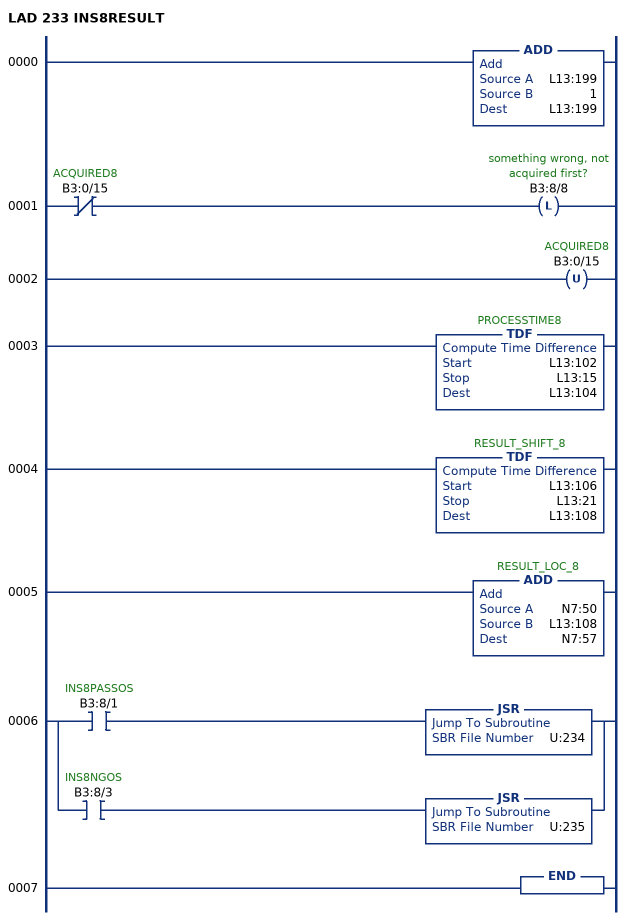
% Rung: 0 %
SOR ADD L13:199 1 L13:199 EOR
% Rung: 1 %
SOR XIO B3:0/15 OTL B3:8/8 EOR
%   B3:0/15  ACQUIRED8 %
%   B3:8/8  "something wrong, not acquired first?" %
% Rung: 2 %
SOR OTU B3:0/15 EOR
%   B3:0/15  ACQUIRED8 %
% Rung: 3 %
SOR TDF L13:102 L13:15 L13:104 EOR
%   L13:102  TIMEOFACQ8 %
%   L13:15  TOP_TIME %
%   L13:104  PROCESSTIME8 %
% Rung: 4 %
SOR TDF L13:106 L13:21 L13:108 EOR
%   L13:106  PROCESS_START_POS_8 %
%   L13:21  TOP_POSITION %
%   L13:108  RESULT_SHIFT_8 %
% Rung: 5 %
SOR ADD N7:50 L13:108 N7:57 EOR
%   N7:50  INS_8_TRIG_LOC %
%   L13:108  RESULT_SHIFT_8 %
%   N7:57  RESULT_LOC_8 %
% Rung: 6 %
SOR BST XIC B3:8/1 JSR U:234 NXB XIC B3:8/3 JSR U:235 BND EOR
%   B3:8/1  INS8PASSOS %
%   B3:8/3  INS8NGOS %
% Rung: 7 %
SOR END EOR

LADDER 234 "INS8PASS"
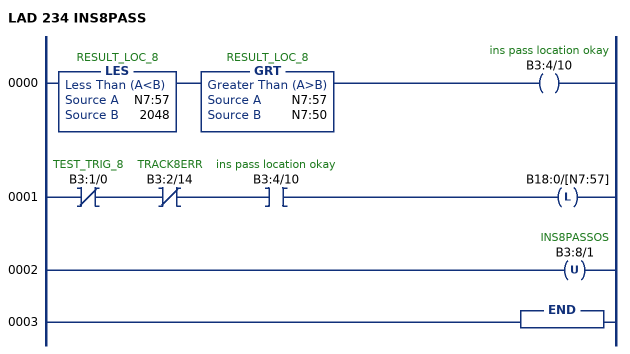
% Rung: 0 %
SOR LES N7:57 2048 GRT N7:57 N7:50 OTE B3:4/10 EOR
%   N7:57  RESULT_LOC_8 %
%   N7:50  INS_8_TRIG_LOC %
%   B3:4/10  "ins pass location okay" %
% Rung: 1 %
SOR XIO B3:1/0 XIO B3:2/14 XIC B3:4/10 OTL B18:0/[N7:57] EOR
%   B3:1/0  TEST_TRIG_8 %
%   B3:2/14  TRACK8ERR %
%   B3:4/10  "ins pass location okay" %
%   B18:0  GOOD2 %
%   N7:57  RESULT_LOC_8 %
% Rung: 2 %
SOR OTU B3:8/1 EOR
%   B3:8/1  INS8PASSOS %
% Rung: 3 %
SOR END EOR

LADDER 235 "INS8FAIL"
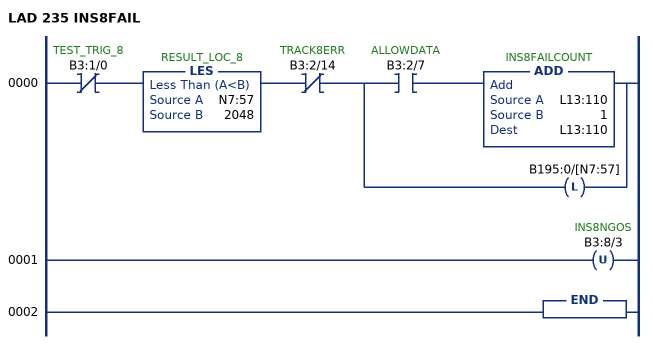
% Rung: 0 %
SOR XIO B3:1/0 LES N7:57 2048 XIO B3:2/14 BST XIC B3:2/7 ADD L13:110 1 L13:110 NXB OTL B195:0/[N7:57] BND EOR
%   B3:1/0  TEST_TRIG_8 %
%   N7:57  RESULT_LOC_8 %
%   B3:2/14  TRACK8ERR %
%   B3:2/7  ALLOWDATA %
%   L13:110  INS8FAILCOUNT %
%   B195:0  TOP_NG %
% Rung: 1 %
SOR OTU B3:8/3 EOR
%   B3:8/3  INS8NGOS %
% Rung: 2 %
SOR END EOR

LADDER 236 "INS8ACQ"
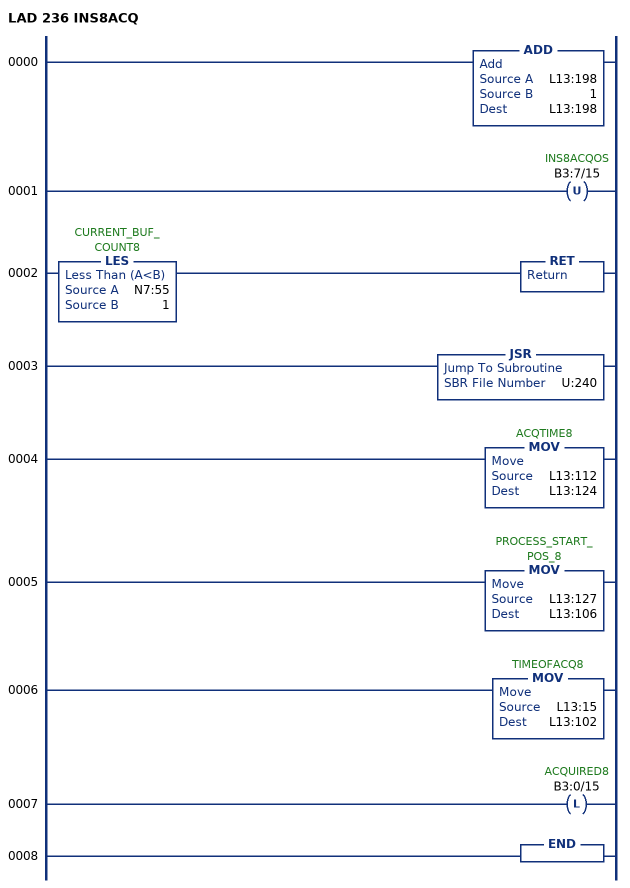
% Rung: 0 %
SOR ADD L13:198 1 L13:198 EOR
% Rung: 1 %
SOR OTU B3:7/15 EOR
%   B3:7/15  INS8ACQOS %
% Rung: 2 %
SOR LES N7:55 1 RET EOR
%   N7:55  CURRENT_BUF_COUNT8 %
% Rung: 3 %
SOR JSR U:240 EOR
% Rung: 4 %
SOR MOV L13:112 L13:124 EOR
%   L13:112  TIME_SPAN8 %
%   L13:124  ACQTIME8 %
% Rung: 5 %
SOR MOV L13:127 L13:106 EOR
%   L13:127  PULLED_POSITION8 %
%   L13:106  PROCESS_START_POS_8 %
% Rung: 6 %
SOR MOV L13:15 L13:102 EOR
%   L13:15  TOP_TIME %
%   L13:102  TIMEOFACQ8 %
% Rung: 7 %
SOR OTL B3:0/15 EOR
%   B3:0/15  ACQUIRED8 %
% Rung: 8 %
SOR END EOR

LADDER 237 "Q8TIMETEST"
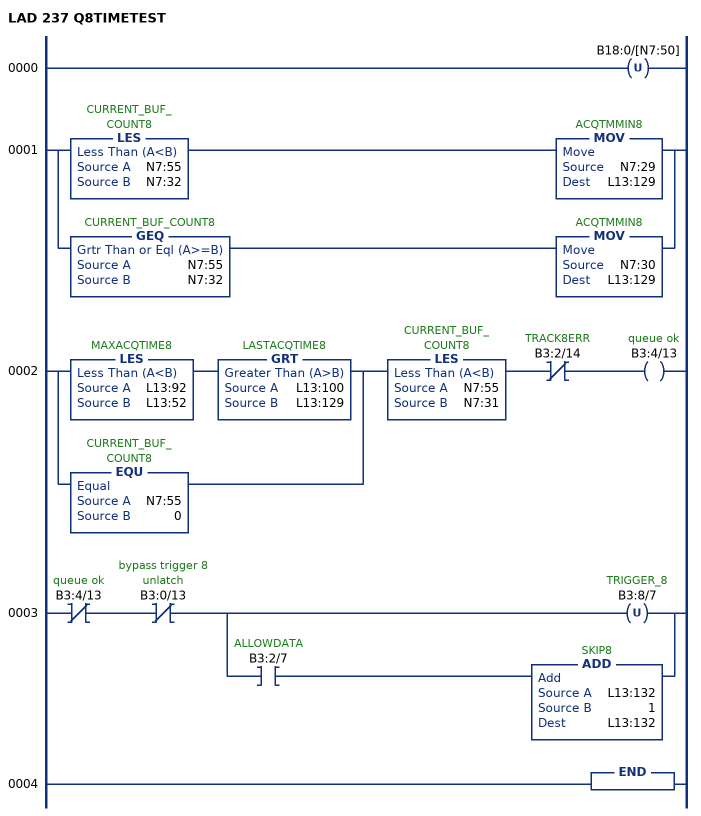
% Rung: 0 %
SOR OTU B18:0/[N7:50] EOR
%   B18:0  GOOD2 %
%   N7:50  INS_8_TRIG_LOC %
% Rung: 1 %
SOR BST LES N7:55 N7:32 MOV N7:29 L13:129 NXB GEQ N7:55 N7:32 MOV N7:30 L13:129 BND EOR
%   N7:55  CURRENT_BUF_COUNT8 %
%   N7:32  BUF_CAM_LIMIT %
%   N7:29  CAM_BUF_ACQ_TM %
%   L13:129  ACQTMMIN8 %
%   N7:30  PC_BUF_ACQ_TM %
% Rung: 2 %
SOR BST LES L13:92 L13:52 GRT L13:100 L13:129 NXB EQU N7:55 0 BND LES N7:55 N7:31 XIO B3:2/14 OTE B3:4/13 EOR
%   L13:92  MAXACQTIME8 %
%   L13:52  ACQTIMELIMIT %
%   L13:100  LASTACQTIME8 %
%   L13:129  ACQTMMIN8 %
%   N7:55  CURRENT_BUF_COUNT8 %
%   N7:31  MAX_BUFF_CT  "maximum buffers" %
%   B3:2/14  TRACK8ERR %
%   B3:4/13  "queue ok" %
% Rung: 3 %
SOR XIO B3:4/13 XIO B3:0/13 BST OTU B3:8/7 NXB XIC B3:2/7 ADD L13:132 1 L13:132 BND EOR
%   B3:4/13  "queue ok" %
%   B3:0/13  "bypass trigger 8 unlatch" %
%   B3:8/7  TRIGGER_8 %
%   B3:2/7  ALLOWDATA %
%   L13:132  SKIP8 %
% Rung: 4 %
SOR END EOR

LADDER 238 "INS8TRIG"
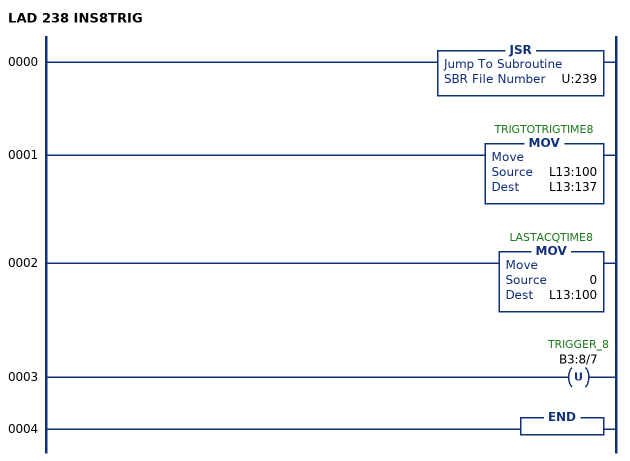
% Rung: 0 %
SOR JSR U:239 EOR
% Rung: 1 %
SOR MOV L13:100 L13:137 EOR
%   L13:100  LASTACQTIME8 %
%   L13:137  TRIGTOTRIGTIME8 %
% Rung: 2 %
SOR MOV 0 L13:100 EOR
%   L13:100  LASTACQTIME8 %
% Rung: 3 %
SOR OTU B3:8/7 EOR
%   B3:8/7  TRIGGER_8 %
% Rung: 4 %
SOR END EOR

LADDER 239 "FIFO8SET"
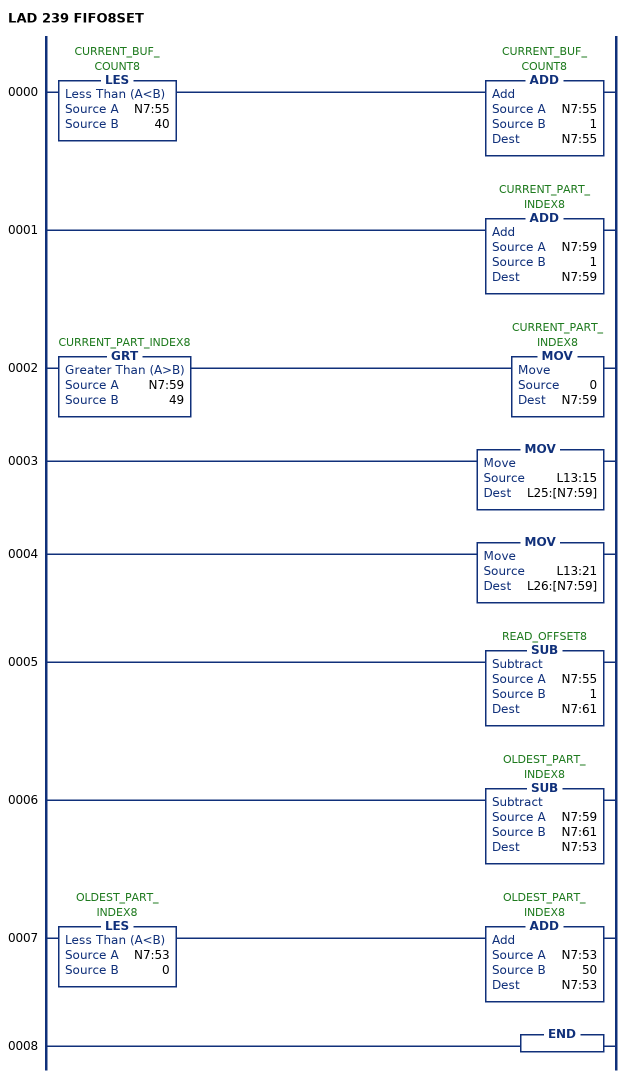
% Rung: 0 %
SOR LES N7:55 40 ADD N7:55 1 N7:55 EOR
%   N7:55  CURRENT_BUF_COUNT8 %
% Rung: 1 %
SOR ADD N7:59 1 N7:59 EOR
%   N7:59  CURRENT_PART_INDEX8 %
% Rung: 2 %
SOR GRT N7:59 49 MOV 0 N7:59 EOR
%   N7:59  CURRENT_PART_INDEX8 %
% Rung: 3 %
SOR MOV L13:15 L25:[N7:59] EOR
%   L13:15  TOP_TIME %
%   N7:59  CURRENT_PART_INDEX8 %
% Rung: 4 %
SOR MOV L13:21 L26:[N7:59] EOR
%   L13:21  TOP_POSITION %
%   N7:59  CURRENT_PART_INDEX8 %
% Rung: 5 %
SOR SUB N7:55 1 N7:61 EOR
%   N7:55  CURRENT_BUF_COUNT8 %
%   N7:61  READ_OFFSET8 %
% Rung: 6 %
SOR SUB N7:59 N7:61 N7:53 EOR
%   N7:59  CURRENT_PART_INDEX8 %
%   N7:61  READ_OFFSET8 %
%   N7:53  OLDEST_PART_INDEX8 %
% Rung: 7 %
SOR LES N7:53 0 ADD N7:53 50 N7:53 EOR
%   N7:53  OLDEST_PART_INDEX8 %
% Rung: 8 %
SOR END EOR

LADDER 240 "FIFO8GET"
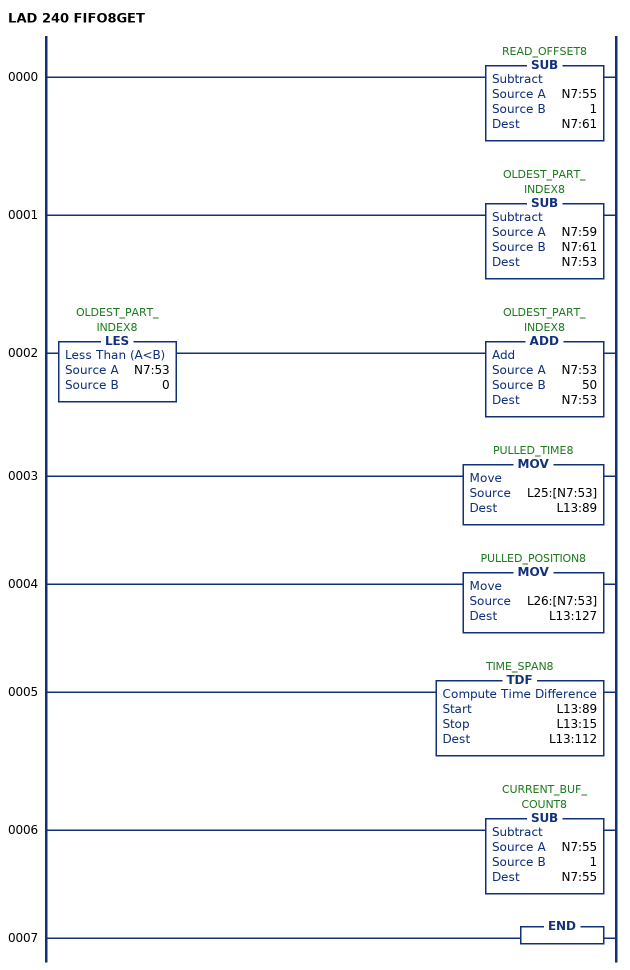
% Rung: 0 %
SOR SUB N7:55 1 N7:61 EOR
%   N7:55  CURRENT_BUF_COUNT8 %
%   N7:61  READ_OFFSET8 %
% Rung: 1 %
SOR SUB N7:59 N7:61 N7:53 EOR
%   N7:59  CURRENT_PART_INDEX8 %
%   N7:61  READ_OFFSET8 %
%   N7:53  OLDEST_PART_INDEX8 %
% Rung: 2 %
SOR LES N7:53 0 ADD N7:53 50 N7:53 EOR
%   N7:53  OLDEST_PART_INDEX8 %
% Rung: 3 %
SOR MOV L25:[N7:53] L13:89 EOR
%   N7:53  OLDEST_PART_INDEX8 %
%   L13:89  PULLED_TIME8 %
% Rung: 4 %
SOR MOV L26:[N7:53] L13:127 EOR
%   N7:53  OLDEST_PART_INDEX8 %
%   L13:127  PULLED_POSITION8 %
% Rung: 5 %
SOR TDF L13:89 L13:15 L13:112 EOR
%   L13:89  PULLED_TIME8 %
%   L13:15  TOP_TIME %
%   L13:112  TIME_SPAN8 %
% Rung: 6 %
SOR SUB N7:55 1 N7:55 EOR
%   N7:55  CURRENT_BUF_COUNT8 %
% Rung: 7 %
SOR END EOR

LADDER 241 "INSDATA8"
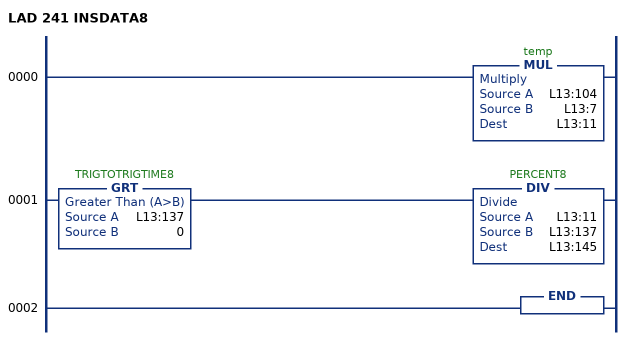
% Rung: 0 %
SOR MUL L13:104 L13:7 L13:11 EOR
%   L13:104  PROCESSTIME8 %
%   L13:7  PERCENT_MULTIPLYER %
%   L13:11  "temp" %
% Rung: 1 %
SOR GRT L13:137 0 DIV L13:11 L13:137 L13:145 EOR
%   L13:137  TRIGTOTRIGTIME8 %
%   L13:11  "temp" %
%   L13:145  PERCENT8 %
% Rung: 2 %
SOR END EOR

LADDER 242 "TESTFAULT8"
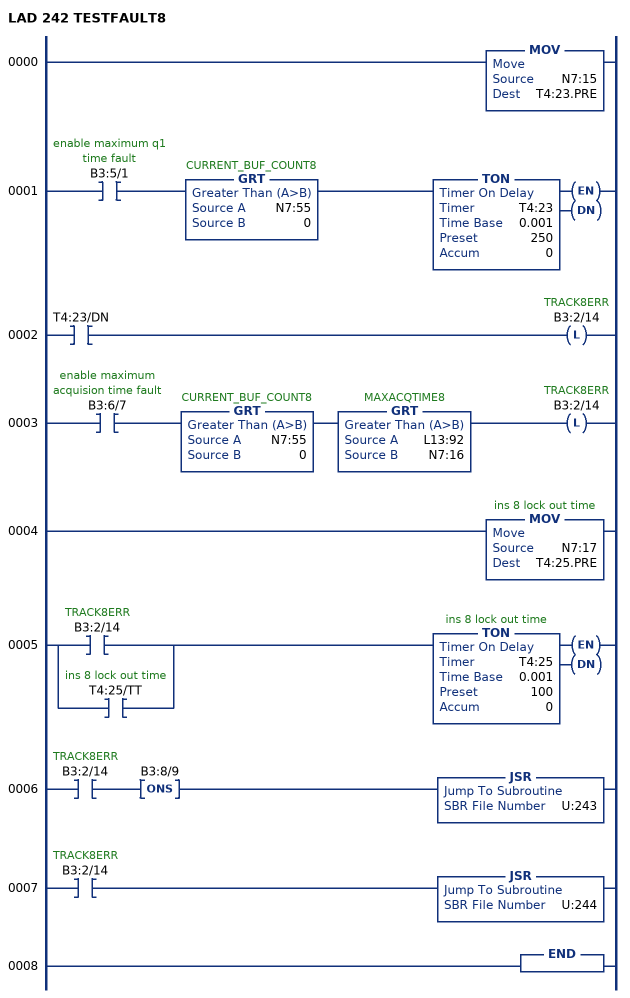
% Rung: 0 %
SOR MOV N7:15 T4:23.PRE EOR
%   N7:15  "max allowed ms time for q to be above 1 if safe fault is used" %
% Rung: 1 %
SOR XIC B3:5/1 GRT N7:55 0 TON T4:23 0.001 250 0 EOR
%   B3:5/1  "enable maximum q1 time fault" %
%   N7:55  CURRENT_BUF_COUNT8 %
% Rung: 2 %
SOR XIC T4:23/DN OTL B3:2/14 EOR
%   B3:2/14  TRACK8ERR %
% Rung: 3 %
SOR XIC B3:6/7 GRT N7:55 0 GRT L13:92 N7:16 OTL B3:2/14 EOR
%   B3:6/7  "enable maximum acquision time fault" %
%   N7:55  CURRENT_BUF_COUNT8 %
%   L13:92  MAXACQTIME8 %
%   N7:16  ACQUIRE_TIME_LIMIT  "maximum of the longest acquire time allowed if maximum acquire time fault is enabled" %
%   B3:2/14  TRACK8ERR %
% Rung: 4 %
SOR MOV N7:17 T4:25.PRE EOR
%   N7:17  "ms time setting to lock out inspection to give all pending images a chance to clear" %
%   T4:25  "ins 8 lock out time" %
% Rung: 5 %
SOR BST XIC B3:2/14 NXB XIC T4:25/TT BND TON T4:25 0.001 100 0 EOR
%   B3:2/14  TRACK8ERR %
%   T4:25  "ins 8 lock out time" %
% Rung: 6 %
SOR XIC B3:2/14 ONS B3:8/9 JSR U:243 EOR
%   B3:2/14  TRACK8ERR %
% Rung: 7 %
SOR XIC B3:2/14 JSR U:244 EOR
%   B3:2/14  TRACK8ERR %
% Rung: 8 %
SOR END EOR

LADDER 243 "INS8FIX1"
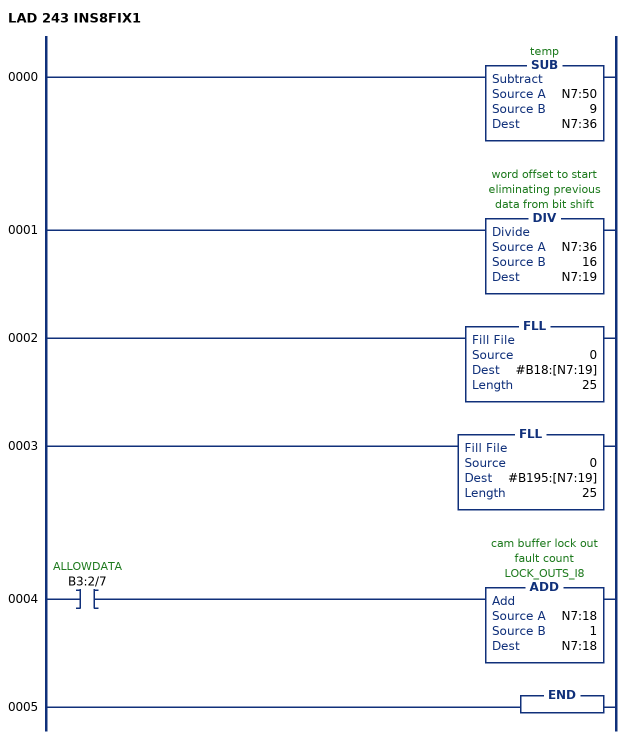
% Rung: 0 %
SOR SUB N7:50 9 N7:36 EOR
%   N7:50  INS_8_TRIG_LOC %
%   N7:36  "temp" %
% Rung: 1 %
SOR DIV N7:36 16 N7:19 EOR
%   N7:36  "temp" %
%   N7:19  "word offset to start eliminating previous data from bit shift" %
% Rung: 2 %
SOR FLL 0 #B18:[N7:19] 25 EOR
%   N7:19  "word offset to start eliminating previous data from bit shift" %
% Rung: 3 %
SOR FLL 0 #B195:[N7:19] 25 EOR
%   N7:19  "word offset to start eliminating previous data from bit shift" %
% Rung: 4 %
SOR XIC B3:2/7 ADD N7:18 1 N7:18 EOR
%   B3:2/7  ALLOWDATA %
%   N7:18  LOCK_OUTS_I8  "cam buffer lock out fault count" %
% Rung: 5 %
SOR END EOR

LADDER 244 "INS8FIX2"
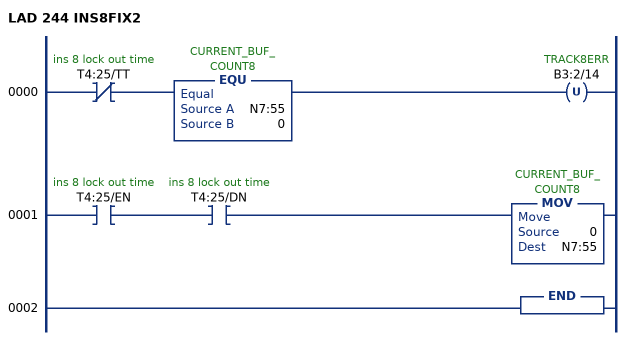
% Rung: 0 %
SOR XIO T4:25/TT EQU N7:55 0 OTU B3:2/14 EOR
%   T4:25  "ins 8 lock out time" %
%   N7:55  CURRENT_BUF_COUNT8 %
%   B3:2/14  TRACK8ERR %
% Rung: 1 %
SOR XIC T4:25/EN XIC T4:25/DN MOV 0 N7:55 EOR
%   T4:25  "ins 8 lock out time" %
%   N7:55  CURRENT_BUF_COUNT8 %
% Rung: 2 %
SOR END EOR

LADDER 249 "PASS BLOW"
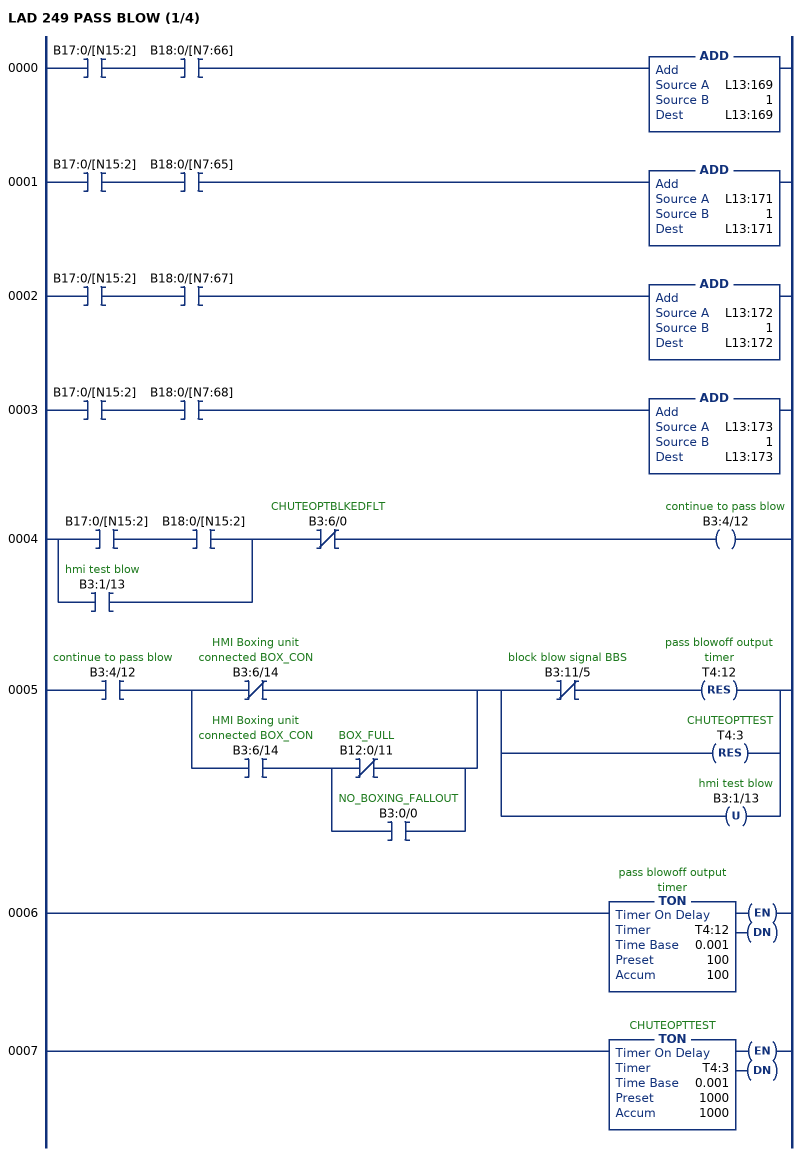
% Rung: 0 %
SOR XIC B17:0/[N15:2] XIC B18:0/[N7:66] ADD L13:169 1 L13:169 EOR
%   B17:0  GOOD1 %
%   N15:2  BLOW_PT %
%   B18:0  GOOD2 %
%   N7:66  P2 %
% Rung: 1 %
SOR XIC B17:0/[N15:2] XIC B18:0/[N7:65] ADD L13:171 1 L13:171 EOR
%   B17:0  GOOD1 %
%   N15:2  BLOW_PT %
%   B18:0  GOOD2 %
%   N7:65  P1 %
% Rung: 2 %
SOR XIC B17:0/[N15:2] XIC B18:0/[N7:67] ADD L13:172 1 L13:172 EOR
%   B17:0  GOOD1 %
%   N15:2  BLOW_PT %
%   B18:0  GOOD2 %
%   N7:67  M1 %
% Rung: 3 %
SOR XIC B17:0/[N15:2] XIC B18:0/[N7:68] ADD L13:173 1 L13:173 EOR
%   B17:0  GOOD1 %
%   N15:2  BLOW_PT %
%   B18:0  GOOD2 %
%   N7:68  M2 %
% Rung: 4 %
SOR BST XIC B17:0/[N15:2] XIC B18:0/[N15:2] NXB XIC B3:1/13 BND XIO B3:6/0 OTE B3:4/12 EOR
%   B17:0  GOOD1 %
%   N15:2  BLOW_PT %
%   B18:0  GOOD2 %
%   B3:1/13  "hmi test blow" %
%   B3:6/0  CHUTEOPTBLKEDFLT %
%   B3:4/12  "continue to pass blow" %
% Rung: 5 %
SOR XIC B3:4/12 BST XIO B3:6/14 NXB XIC B3:6/14 BST XIO B12:0/11 NXB XIC B3:0/0 BND BND BST XIO B3:11/5 RES T4:12 NXB RES T4:3 NXB OTU B3:1/13 BND EOR
%   B3:4/12  "continue to pass blow" %
%   B3:6/14  BOX_CON  "HMI Boxing unit connected" %
%   B12:0/11  BOX_FULL %
%   B3:0/0  NO_BOXING_FALLOUT %
%   B3:11/5  BBS  "block blow signal" %
%   T4:12  "pass blowoff output timer" %
%   T4:3  CHUTEOPTTEST %
%   B3:1/13  "hmi test blow" %
% Rung: 6 %
SOR TON T4:12 0.001 100 100 EOR
%   T4:12  "pass blowoff output timer" %
% Rung: 7 %
SOR TON T4:3 0.001 1000 1000 EOR
%   T4:3  CHUTEOPTTEST %

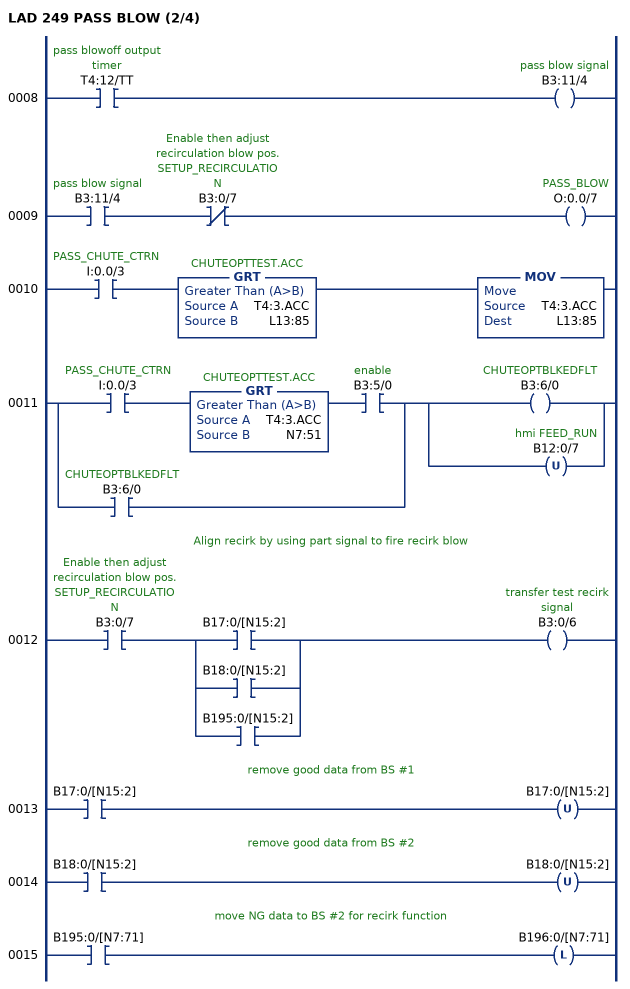
% Rung: 8 %
SOR XIC T4:12/TT OTE B3:11/4 EOR
%   T4:12  "pass blowoff output timer" %
%   B3:11/4  "pass blow signal" %
% Rung: 9 %
SOR XIC B3:11/4 XIO B3:0/7 OTE O:0.0/7 EOR
%   B3:11/4  "pass blow signal" %
%   B3:0/7  SETUP_RECIRCULATION  "Enable then adjust recirculation blow pos." %
%   O:0.0/7  PASS_BLOW %
% Rung: 10 %
SOR XIC I:0.0/3 GRT T4:3.ACC L13:85 MOV T4:3.ACC L13:85 EOR
%   I:0.0/3  PASS_CHUTE_CTRN %
%   T4:3  CHUTEOPTTEST %
% Rung: 11 %
SOR BST XIC I:0.0/3 GRT T4:3.ACC N7:51 XIC B3:5/0 NXB XIC B3:6/0 BND BST OTE B3:6/0 NXB OTU B12:0/7 BND EOR
%   I:0.0/3  PASS_CHUTE_CTRN %
%   T4:3  CHUTEOPTTEST %
%   B3:5/0  "enable" %
%   B3:6/0  CHUTEOPTBLKEDFLT %
%   B12:0/7  FEED_RUN  "hmi" %
% Rung: 12 %
% Align recirk by using part signal to fire recirk blow %
SOR XIC B3:0/7 BST XIC B17:0/[N15:2] NXB XIC B18:0/[N15:2] NXB XIC B195:0/[N15:2] BND OTE B3:0/6 EOR
%   B3:0/7  SETUP_RECIRCULATION  "Enable then adjust recirculation blow pos." %
%   B17:0  GOOD1 %
%   N15:2  BLOW_PT %
%   B18:0  GOOD2 %
%   B195:0  TOP_NG %
%   B3:0/6  "transfer test recirk signal" %
% Rung: 13 %
% remove good data from BS #1 %
SOR XIC B17:0/[N15:2] OTU B17:0/[N15:2] EOR
%   B17:0  GOOD1 %
%   N15:2  BLOW_PT %
% Rung: 14 %
% remove good data from BS #2 %
SOR XIC B18:0/[N15:2] OTU B18:0/[N15:2] EOR
%   B18:0  GOOD2 %
%   N15:2  BLOW_PT %
% Rung: 15 %
% move NG data to BS #2 for recirk function %
SOR XIC B195:0/[N7:71] OTL B196:0/[N7:71] EOR
%   B195:0  TOP_NG %
%   N7:71  RESIRK_START_BIT %
%   B196:0  RECK_FAIL_TRK %

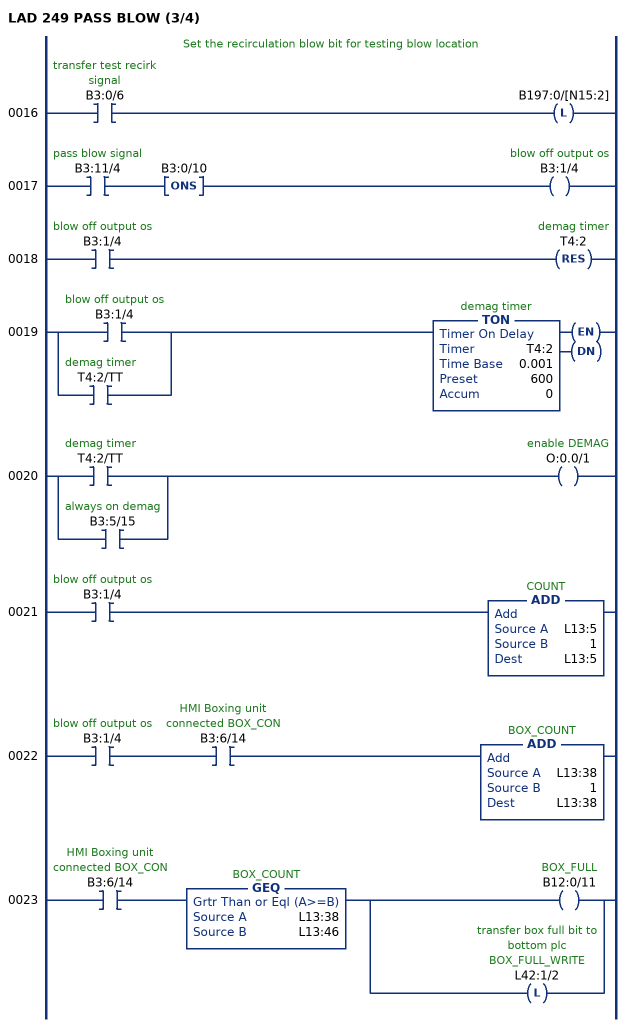
% Rung: 16 %
% Set the recirculation blow bit for testing blow location %
SOR XIC B3:0/6 OTL B197:0/[N15:2] EOR
%   B3:0/6  "transfer test recirk signal" %
%   B197:0  RECK_BLOW_TRK %
%   N15:2  BLOW_PT %
% Rung: 17 %
SOR XIC B3:11/4 ONS B3:0/10 OTE B3:1/4 EOR
%   B3:11/4  "pass blow signal" %
%   B3:1/4  "blow off output os" %
% Rung: 18 %
SOR XIC B3:1/4 RES T4:2 EOR
%   B3:1/4  "blow off output os" %
%   T4:2  "demag timer" %
% Rung: 19 %
SOR BST XIC B3:1/4 NXB XIC T4:2/TT BND TON T4:2 0.001 600 0 EOR
%   B3:1/4  "blow off output os" %
%   T4:2  "demag timer" %
% Rung: 20 %
SOR BST XIC T4:2/TT NXB XIC B3:5/15 BND OTE O:0.0/1 EOR
%   T4:2  "demag timer" %
%   B3:5/15  "always on demag" %
%   O:0.0/1  DEMAG  "enable" %
% Rung: 21 %
SOR XIC B3:1/4 ADD L13:5 1 L13:5 EOR
%   B3:1/4  "blow off output os" %
%   L13:5  COUNT %
% Rung: 22 %
SOR XIC B3:1/4 XIC B3:6/14 ADD L13:38 1 L13:38 EOR
%   B3:1/4  "blow off output os" %
%   B3:6/14  BOX_CON  "HMI Boxing unit connected" %
%   L13:38  BOX_COUNT %
% Rung: 23 %
SOR XIC B3:6/14 GEQ L13:38 L13:46 BST OTE B12:0/11 NXB OTL L42:1/2 BND EOR
%   B3:6/14  BOX_CON  "HMI Boxing unit connected" %
%   L13:38  BOX_COUNT %
%   L13:46  BOX_LIMIT  "box count setpoint" %
%   B12:0/11  BOX_FULL %
%   L42:1/2  BOX_FULL_WRITE  "transfer box full bit to bottom plc" %

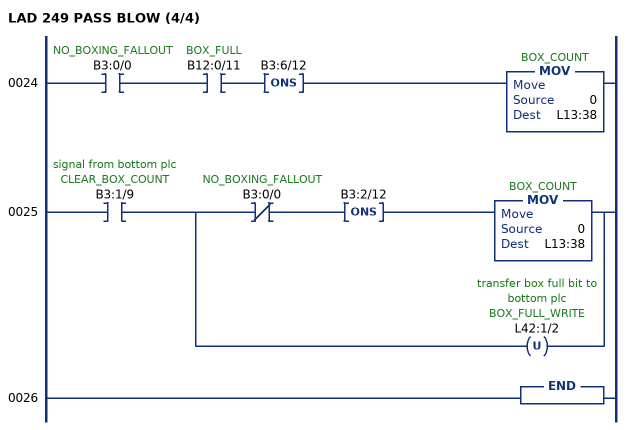
% Rung: 24 %
SOR XIC B3:0/0 XIC B12:0/11 ONS B3:6/12 MOV 0 L13:38 EOR
%   B3:0/0  NO_BOXING_FALLOUT %
%   B12:0/11  BOX_FULL %
%   L13:38  BOX_COUNT %
% Rung: 25 %
SOR XIC B3:1/9 BST XIO B3:0/0 ONS B3:2/12 MOV 0 L13:38 NXB OTU L42:1/2 BND EOR
%   B3:1/9  CLEAR_BOX_COUNT  "signal from bottom plc" %
%   B3:0/0  NO_BOXING_FALLOUT %
%   L13:38  BOX_COUNT %
%   L42:1/2  BOX_FULL_WRITE  "transfer box full bit to bottom plc" %
% Rung: 26 %
SOR END EOR

LADDER 250 "RECIRK"
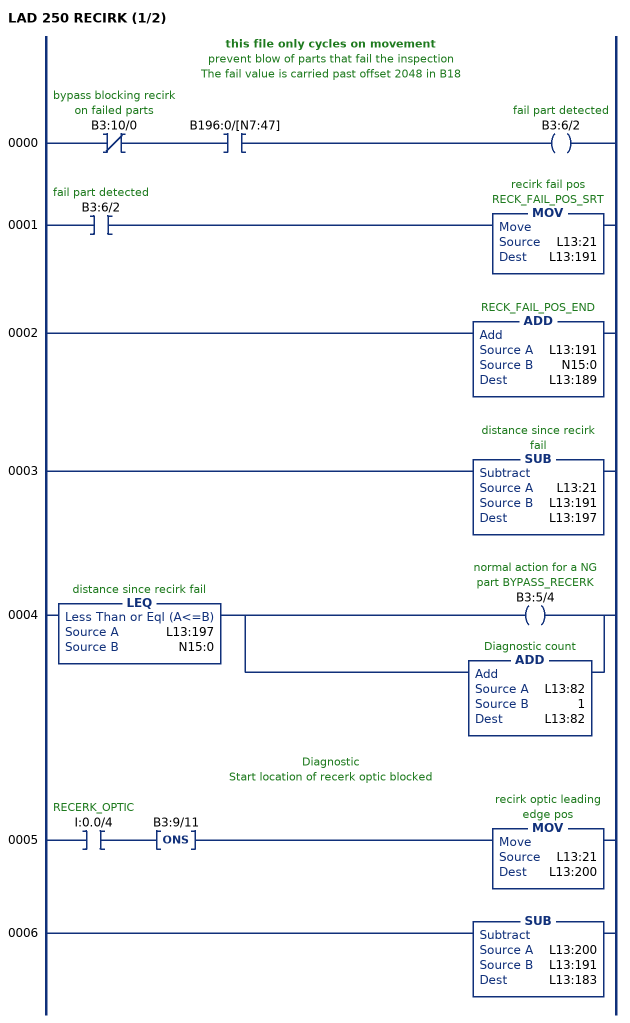
% Rung: 0 %
% TITLE: this file only cycles on movement %
% prevent blow of parts that fail the inspection
% The fail value is carried past offset 2048 in B18 %
SOR XIO B3:10/0 XIC B196:0/[N7:47] OTE B3:6/2 EOR
%   B3:10/0  "bypass blocking recirk on failed parts" %
%   B196:0  RECK_FAIL_TRK %
%   N7:47  RECERK_BLOCKOPTIC_PT %
%   B3:6/2  "fail part detected" %
% Rung: 1 %
SOR XIC B3:6/2 MOV L13:21 L13:191 EOR
%   B3:6/2  "fail part detected" %
%   L13:21  TOP_POSITION %
%   L13:191  RECK_FAIL_POS_SRT  "recirk fail pos" %
% Rung: 2 %
SOR ADD L13:191 N15:0 L13:189 EOR
%   L13:191  RECK_FAIL_POS_SRT  "recirk fail pos" %
%   N15:0  RECIRK_FAIL_ZONE  "Recirculation fail zone width" %
%   L13:189  RECK_FAIL_POS_END %
% Rung: 3 %
SOR SUB L13:21 L13:191 L13:197 EOR
%   L13:21  TOP_POSITION %
%   L13:191  RECK_FAIL_POS_SRT  "recirk fail pos" %
%   L13:197  "distance since recirk fail" %
% Rung: 4 %
SOR LEQ L13:197 N15:0 BST OTE B3:5/4 NXB ADD L13:82 1 L13:82 BND EOR
%   L13:197  "distance since recirk fail" %
%   N15:0  RECIRK_FAIL_ZONE  "Recirculation fail zone width" %
%   B3:5/4  BYPASS_RECERK  "normal action for a NG part" %
%   L13:82  "Diagnostic count" %
% Rung: 5 %
% Diagnostic
% Start location of recerk optic blocked %
SOR XIC I:0.0/4 ONS B3:9/11 MOV L13:21 L13:200 EOR
%   I:0.0/4  RECERK_OPTIC %
%   L13:21  TOP_POSITION %
%   L13:200  "recirk optic leading edge pos" %
% Rung: 6 %
SOR SUB L13:200 L13:191 L13:183 EOR
%   L13:200  "recirk optic leading edge pos" %
%   L13:191  RECK_FAIL_POS_SRT  "recirk fail pos" %

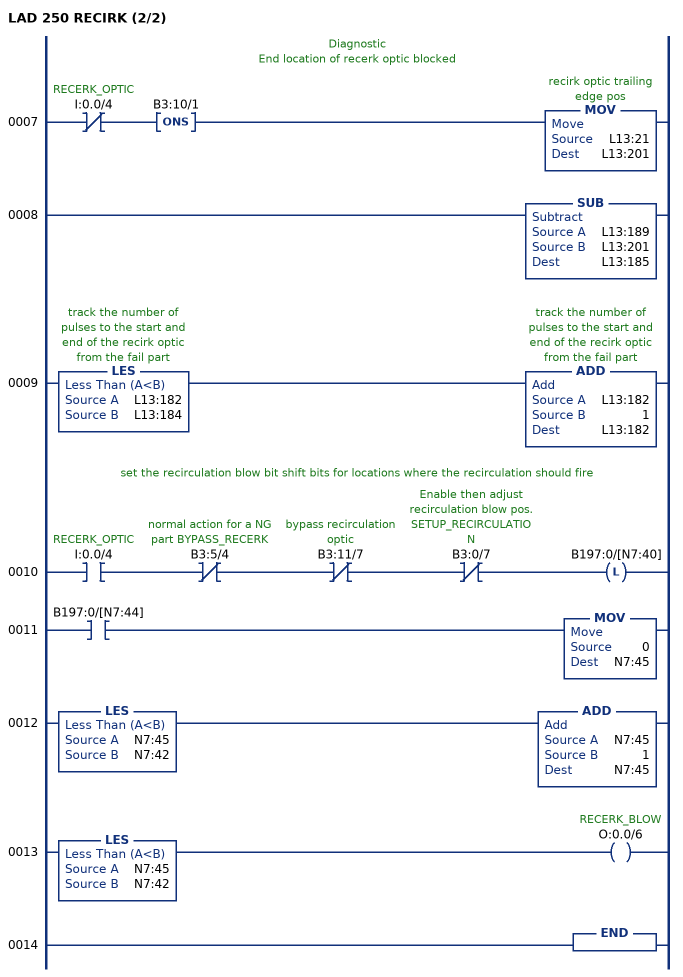
% Rung: 7 %
% Diagnostic
% End location of recerk optic blocked %
SOR XIO I:0.0/4 ONS B3:10/1 MOV L13:21 L13:201 EOR
%   I:0.0/4  RECERK_OPTIC %
%   L13:21  TOP_POSITION %
%   L13:201  "recirk optic trailing edge pos" %
% Rung: 8 %
SOR SUB L13:189 L13:201 L13:185 EOR
%   L13:189  RECK_FAIL_POS_END %
%   L13:201  "recirk optic trailing edge pos" %
% Rung: 9 %
SOR LES L13:182 L13:184 ADD L13:182 1 L13:182 EOR
%   L13:182  "track the number of pulses to the start and end of the recirk optic from the fail part" %
% Rung: 10 %
% set the recirculation blow bit shift bits for locations where the recirculation should fire %
SOR XIC I:0.0/4 XIO B3:5/4 XIO B3:11/7 XIO B3:0/7 OTL B197:0/[N7:40] EOR
%   I:0.0/4  RECERK_OPTIC %
%   B3:5/4  BYPASS_RECERK  "normal action for a NG part" %
%   B3:11/7  "bypass recirculation optic" %
%   B3:0/7  SETUP_RECIRCULATION  "Enable then adjust recirculation blow pos." %
%   B197:0  RECK_BLOW_TRK %
%   N7:40  RECERK_OPTIC_POS %
% Rung: 11 %
SOR XIC B197:0/[N7:44] MOV 0 N7:45 EOR
%   B197:0  RECK_BLOW_TRK %
%   N7:44  RECERK_BLOW_POS  "adjusted for blow length" %
% Rung: 12 %
SOR LES N7:45 N7:42 ADD N7:45 1 N7:45 EOR
%   N7:42  RECIRK_WIDTH %
% Rung: 13 %
SOR LES N7:45 N7:42 OTE O:0.0/6 EOR
%   N7:42  RECIRK_WIDTH %
%   O:0.0/6  RECERK_BLOW %
% Rung: 14 %
SOR END EOR

LADDER 251 "RECIRK SET"
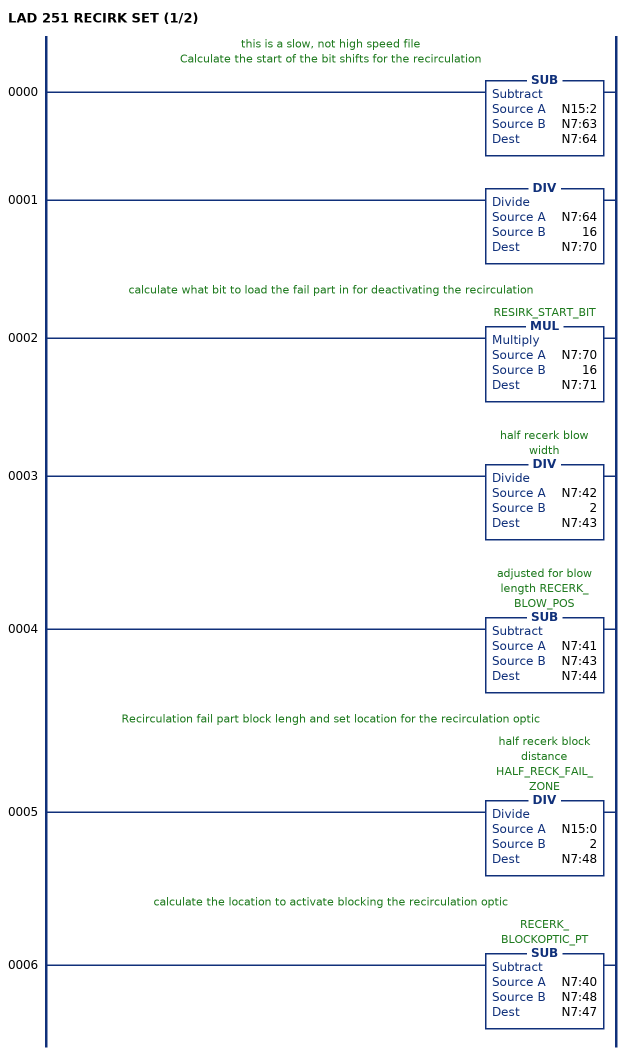
% Rung: 0 %
% this is a slow, not high speed file
% 
% Calculate the start of the bit shifts for the recirculation %
SOR SUB N15:2 N7:63 N7:64 EOR
%   N15:2  BLOW_PT %
% Rung: 1 %
SOR DIV N7:64 16 N7:70 EOR
% Rung: 2 %
% calculate what bit to load the fail part in for deactivating the recirculation %
SOR MUL N7:70 16 N7:71 EOR
%   N7:71  RESIRK_START_BIT %
% Rung: 3 %
SOR DIV N7:42 2 N7:43 EOR
%   N7:42  RECIRK_WIDTH %
%   N7:43  "half recerk blow width" %
% Rung: 4 %
SOR SUB N7:41 N7:43 N7:44 EOR
%   N7:41  RECERK_BLOW_POS_HMI  "recerk blow position set from hmi" %
%   N7:43  "half recerk blow width" %
%   N7:44  RECERK_BLOW_POS  "adjusted for blow length" %
% Rung: 5 %
% Recirculation fail part block lengh and set location for the recirculation optic %
SOR DIV N15:0 2 N7:48 EOR
%   N15:0  RECIRK_FAIL_ZONE  "Recirculation fail zone width" %
%   N7:48  HALF_RECK_FAIL_ZONE  "half recerk block distance" %
% Rung: 6 %
% calculate the location to activate blocking the recirculation optic %
SOR SUB N7:40 N7:48 N7:47 EOR
%   N7:40  RECERK_OPTIC_POS %
%   N7:48  HALF_RECK_FAIL_ZONE  "half recerk block distance" %
%   N7:47  RECERK_BLOCKOPTIC_PT %

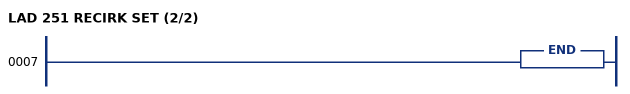
% Rung: 7 %
SOR END EOR

LADDER 252 "RATE1"
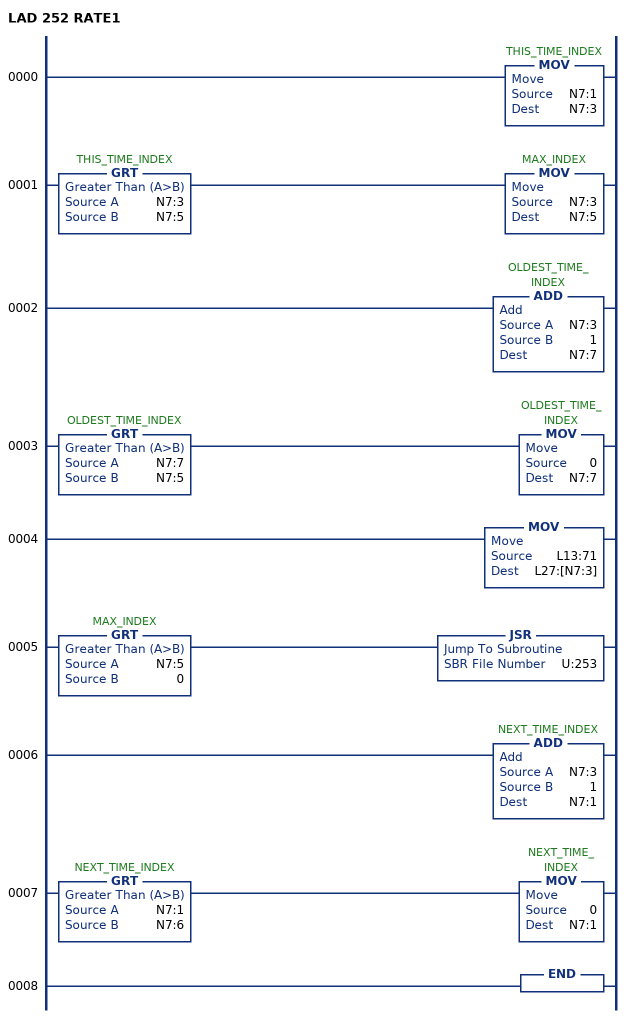
% Rung: 0 %
SOR MOV N7:1 N7:3 EOR
%   N7:1  NEXT_TIME_INDEX %
%   N7:3  THIS_TIME_INDEX %
% Rung: 1 %
SOR GRT N7:3 N7:5 MOV N7:3 N7:5 EOR
%   N7:3  THIS_TIME_INDEX %
%   N7:5  MAX_INDEX %
% Rung: 2 %
SOR ADD N7:3 1 N7:7 EOR
%   N7:3  THIS_TIME_INDEX %
%   N7:7  OLDEST_TIME_INDEX %
% Rung: 3 %
SOR GRT N7:7 N7:5 MOV 0 N7:7 EOR
%   N7:7  OLDEST_TIME_INDEX %
%   N7:5  MAX_INDEX %
% Rung: 4 %
SOR MOV L13:71 L27:[N7:3] EOR
%   L13:71  HSC_TIME %
%   N7:3  THIS_TIME_INDEX %
% Rung: 5 %
SOR GRT N7:5 0 JSR U:253 EOR
%   N7:5  MAX_INDEX %
% Rung: 6 %
SOR ADD N7:3 1 N7:1 EOR
%   N7:3  THIS_TIME_INDEX %
%   N7:1  NEXT_TIME_INDEX %
% Rung: 7 %
SOR GRT N7:1 N7:6 MOV 0 N7:1 EOR
%   N7:1  NEXT_TIME_INDEX %
%   N7:6  UPPER_INDEX_LIMIT  "buffer count 1" %
% Rung: 8 %
SOR END EOR

LADDER 253 "RATE2"
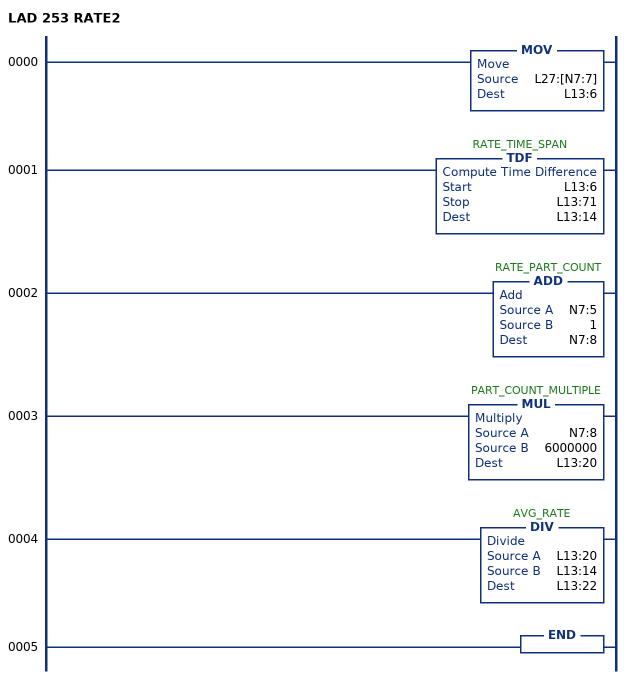
% Rung: 0 %
SOR MOV L27:[N7:7] L13:6 EOR
%   N7:7  OLDEST_TIME_INDEX %
% Rung: 1 %
SOR TDF L13:6 L13:71 L13:14 EOR
%   L13:71  HSC_TIME %
%   L13:14  RATE_TIME_SPAN %
% Rung: 2 %
SOR ADD N7:5 1 N7:8 EOR
%   N7:5  MAX_INDEX %
%   N7:8  RATE_PART_COUNT %
% Rung: 3 %
SOR MUL N7:8 6000000 L13:20 EOR
%   N7:8  RATE_PART_COUNT %
%   L13:20  PART_COUNT_MULTIPLE %
% Rung: 4 %
SOR DIV L13:20 L13:14 L13:22 EOR
%   L13:20  PART_COUNT_MULTIPLE %
%   L13:14  RATE_TIME_SPAN %
%   L13:22  AVG_RATE %
% Rung: 5 %
SOR END EOR

LADDER 254 "RESET RATE"
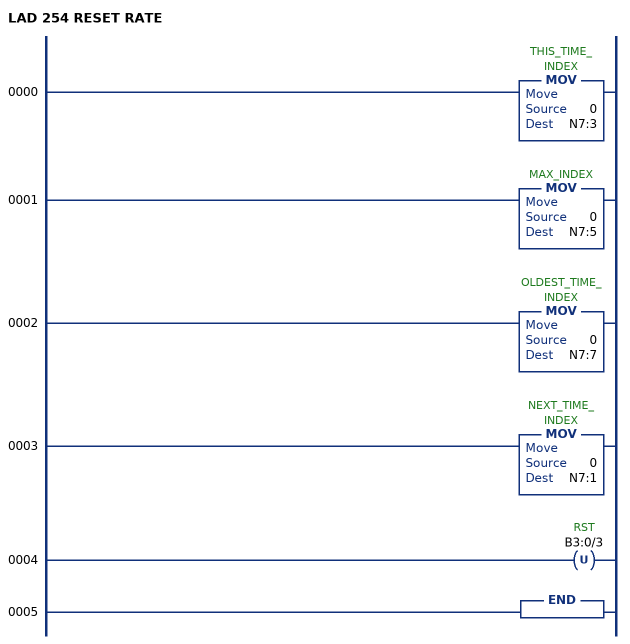
% Rung: 0 %
SOR MOV 0 N7:3 EOR
%   N7:3  THIS_TIME_INDEX %
% Rung: 1 %
SOR MOV 0 N7:5 EOR
%   N7:5  MAX_INDEX %
% Rung: 2 %
SOR MOV 0 N7:7 EOR
%   N7:7  OLDEST_TIME_INDEX %
% Rung: 3 %
SOR MOV 0 N7:1 EOR
%   N7:1  NEXT_TIME_INDEX %
% Rung: 4 %
SOR OTU B3:0/3 EOR
%   B3:0/3  RST %
% Rung: 5 %
SOR END EOR

LADDER 255 "UNUSED"
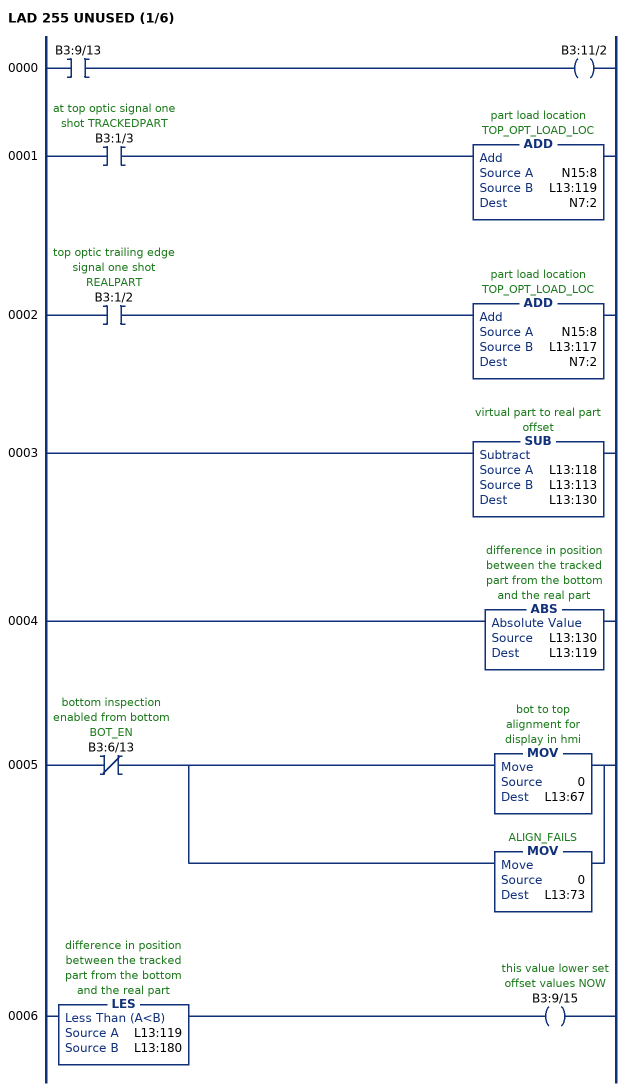
% Rung: 0 %
SOR XIC B3:9/13 OTE B3:11/2 EOR
% Rung: 1 %
SOR XIC B3:1/3 ADD N15:8 L13:119 N7:2 EOR
%   B3:1/3  TRACKEDPART  "at top optic signal one shot" %
%   N15:8  TOP_OPTIC_LOC %
%   L13:119  "difference in position between the tracked part from the bottom and the real part" %
%   N7:2  TOP_OPT_LOAD_LOC  "part load location" %
% Rung: 2 %
SOR XIC B3:1/2 ADD N15:8 L13:117 N7:2 EOR
%   B3:1/2  REALPART  "top optic trailing edge signal one shot" %
%   N15:8  TOP_OPTIC_LOC %
%   L13:117  HALF_WIDTH  "1/2 width top" %
%   N7:2  TOP_OPT_LOAD_LOC  "part load location" %
% Rung: 3 %
SOR SUB L13:118 L13:113 L13:130 EOR
%   L13:118  REAL_CL_POSITION  "real part center line in raw position" %
%   L13:113  VERTUAL_CL_POSITION  "virtual part center line transfer from the bottom in raw position" %
%   L13:130  "virtual part to real part offset" %
% Rung: 4 %
SOR ABS L13:130 L13:119 EOR
%   L13:130  "virtual part to real part offset" %
%   L13:119  "difference in position between the tracked part from the bottom and the real part" %
% Rung: 5 %
SOR XIO B3:6/13 BST MOV 0 L13:67 NXB MOV 0 L13:73 BND EOR
%   B3:6/13  BOT_EN  "bottom inspection enabled from bottom" %
%   L13:67  "bot to top alignment for display in hmi" %
%   L13:73  ALIGN_FAILS %
% Rung: 6 %
SOR LES L13:119 L13:180 OTE B3:9/15 EOR
%   L13:119  "difference in position between the tracked part from the bottom and the real part" %
%   L13:180  "last absolute offset" %
%   B3:9/15  NOW  "this value lower set offset values" %

